// TIA Portal V21 export
// export: Created 2026-07-07T09:15:55.8352405Z, ExportSetting WithReadOnly, DisplayName Totally Integrated Automation Portal, DisplayVersion V21, DisplayName SINAMICS Startdrive Advanced, DisplayVersion V21, DisplayName SINAMICS Startdrive G110M, G120, G120C, G120D, G120P, G115D, DisplayVersion V21, DisplayName SINAMICS Startdrive G130, G150, S120, S150, G200, G220, S200, S210, S220, Innomotics MVD, DisplayVersion V21, DisplayName STEP 7 Professional, DisplayVersion V21, DisplayName STEP 7 Safety, DisplayVersion V21, DisplayName Tech WebApplication, DisplayVersion V21, DisplayName WinCC Basic/Comfort/Advanced, DisplayVersion V21, DisplayName WinCC Professional, DisplayVersion V21, DisplayName WinCC Unified, DisplayVersion V21
Screen "Screen_04_AlarmsDiagnostics"  Nonex480, Template=模板_1
  ScreenLayer 
    TextField "Title" at 20,12 size 760x34  Text="画面 4：报警与诊断"
    TextField "NavBar" at 20,430 size 760x34  Text="主监控 手动调试 参数设置 报警诊断 趋势"
    TextField "Hdr_Item_288" at 20,60 size 360x26  Text="报警摘要"
    TextField "Body_Item_304" at 20,84 size 360x96  Text="System_Alarm_Light | Emergency_Stop | Remote_Comms_OK | Comm_Normal"
    TextField "Hdr_Item_320" at 20,190 size 360x26  Text="通信诊断"
    TextField "Body_Item_336" at 20,214 size 360x166  Text="Remote_Heartbeat | Last_Heartbeat | Watchdog_Timer | Watchdog_Count | Remote_Comms_Was_OK"
    TextField "Hdr_Item_352" at 410,60 size 370x26  Text="模式联锁诊断"
    TextField "Body_Item_368" at 410,84 size 370x96  Text="Manual_Mode | Auto_Mode | Manual_Active | Auto_Active | Manual_PumpValve_Enable"
    TextField "Hdr_Item_384" at 410,190 size 370x26  Text="手动执行快照"
    TextField "Body_Item_400" at 410,214 size 370x166  Text="Manual_q_f_Set | Manual_q_f_Selected | Manual_q_a_Set | Manual_q_a_Selected | q_f_cmd | q_a_cmd"
